FUNCTION TryConvert_SINT_TO_TIME : BOOL
VAR_INPUT
	in : SINT;
	out : REFERENCE TO TIME;
END_VAR

IF in < DatatypeLimits.MIN_VALUE_OF_SINT_WHICH_CAN_BE_HELD_IN_A_TIME THEN
	RETURN;
END_IF

out := SINT_TO_TIME(in);
TryConvert_SINT_TO_TIME := TRUE;

END_FUNCTION

(* stored: Version 1.1.0.1, ProductVersion 3.1.4024.12
   POU TryConvert_SINT_TO_TIME: Id {5f7c24bd-de90-4936-90ba-88557b70a5b2}, SpecialFunc None *)
